{attribute 'linkalways'} 
{attribute 'no_explicit_call' := 'This FB is a CLASS and must be accessed using methods or properties'}
{attribute 'enable_dynamic_creation'}
FUNCTION_BLOCK Node_F_VN_InsertIntoContainer_DINT EXTENDS VisionNode
VAR
    nElement : _DINT(0);
    ipContainer : _ITcVnContainer;
    nIndex : _ULINT(0);
    hrPrev : _HRESULT(S_OK);
    hresult : _HRESULT(S_OK);
END_VAR

METHOD PUBLIC  Clone : I_Node
VAR
	pNode : POINTER TO Node_F_VN_InsertIntoContainer_DINT;
END_VAR
pNode := __NEW(Node_F_VN_InsertIntoContainer_DINT);
Clone := pNode^;
END_METHOD

METHOD FB_init : BOOL
VAR_INPUT
	bInitRetains : BOOL; // if TRUE, the retain variables are initialized (warm start / cold start)
	bInCopyCode : BOOL;  // if TRUE, the instance afterwards gets moved into the copy code (online change)
END_VAR
AddInput('nElement', nElement);
AddInput('ipContainer', ipContainer);
AddInput('nIndex', nIndex);
AddInput('hrPrev', hrPrev);
AddOutput('ipContainer', ipContainer);
AddOutput('hresult',hresult);
END_METHOD

METHOD PROTECTED OnExecute : HRESULT
hresult.Value := F_VN_InsertIntoContainer_DINT(
    nElement := nElement.Value,
    ipContainer := ipContainer.Value,
    nIndex := nIndex.Value,
    hrPrev:= hrPrev.Value);
END_METHOD

METHOD PUBLIC PreExecutionCheck
VAR_INPUT
	Check : I_PreExecutionChecks;
END_VAR
Check.IsTrue(ipContainer.IsValid, 'ipContainer must be a valid container');
Check.IsTrue(ipContainer.HasType('CTcVnContainer_Vector_DINT'), 'ipContainer contains incorrect types');
END_METHOD

END_FUNCTION_BLOCK

(* stored: Version 1.1.0.1, ProductVersion 3.1.4024.13
   POU Node_F_VN_InsertIntoContainer_DINT: Id {5c33d4b9-d64b-42e8-b477-6791fd58535b}, SpecialFunc None
   Folder Constructor: Id {5ce73643-52fe-43e0-af25-ea46982e847c}
   Method Clone: Id {6df29656-acb6-4228-b73b-c6dea66a0e11}
   Method FB_init: Id {62d2f1e5-07a5-48e4-b9de-d46189dbdef0}
   Method OnExecute: Id {491c5abd-face-4468-bafd-1d04703837d0}
   Method PreExecutionCheck: Id {a7cff66c-eaf1-43af-88ae-6ec595f8115d} *)
